(* PLC project Programme MGS_2-07_refactorJOY.project, CODESYS CODESYS V3.5 SP19 Patch 1 *)
(* stored: creationDateTime 2026-06-29T23:37:40.2324756, modificationDateTime 2026-06-29T22:49:33.424 *)

FUNCTION_BLOCK FB_CycleTime
  VAR_INPUT
    DefaultValueS : REAL := 0.004;  (* Valeur de secours (Ex: MainTask = 20ms -> 0.020) *)
  END_VAR
  VAR_OUTPUT
    CycleTimeS : REAL;  (* Temps écoulé réel (Secondes) *)
  END_VAR
  VAR
    TimeCurrent : TIME;  (* Temps système actuel *)
    TimeLast : TIME;  (* Empreinte du cycle précédent *)
    DeltaTimeMs : UDINT;  (* Écart brut calculé *)
    InitDone : BOOL;  (* Drapeau d'initialisation *)
  END_VAR

            // 1. ACQUISITION DU TEMPS SYSTÈME
TimeCurrent := TIME();

// 2. INITIALISATION UNIQUE AU PREMIER CYCLE
IF NOT InitDone THEN
    TimeLast := TimeCurrent; // ◄ Fixé ici pour éviter un calcul faussé au cycle 2
    InitDone := TRUE;
    CycleTimeS := DefaultValueS;
    RETURN;
END_IF;

// 3. CALCUL DU DELTA EN MILLISECONDES
DeltaTimeMs := TIME_TO_UDINT(TimeCurrent - TimeLast);

// 4. CONVERSION ET CHARGE DE SECOURS
IF DeltaTimeMs > 0 THEN
    CycleTimeS := UDINT_TO_REAL(DeltaTimeMs) / 1000.0;
ELSE
    CycleTimeS := DefaultValueS;
END_IF;

// 5. ARCHIVAGE POUR LE PROCHAIN CYCLE
TimeLast := TimeCurrent;
          
END_FUNCTION_BLOCK
